       #STATE_DISCONNECTING:
         IF #disconnect.STATUS = #RESULT_JOB_START THEN
           #connectionStatus.isConnected := FALSE;
           #connectionStatus.isDisconnecting := TRUE;

         ELSIF #disconnect.STATUS = #RESULT_IDLE THEN
           #connectionStatus.isDisconnecting := TRUE;
           #disconnect.REQ := NOT #disconnect.REQ;

         ELSIF #disconnect.STATUS = #RESULT_JOB_RUNNING THEN
           #disconnect.REQ := FALSE;

         ELSIF #disconnect.STATUS = #RESULT_JOB_NOT_REQUIRED OR
           #disconnect.STATUS = #RESULT_SUCCESS
         THEN
           #disconnect.REQ := FALSE;
           #connectionStatus.isConnected := FALSE;
           #connectionStatus.isDisconnecting := FALSE;
           #connectionStatus.isDisconnected := TRUE;
           #connectionStatus.hasReceivedData := FALSE;
           #connectionStatus.hasReceivedHeader := FALSE;

           #ownInstance := 0;
           #ownSequence := 0;
           #Config.connID := 0;

           #internalState := #STATE_IDLE;
         ELSE
           // Throw error !
           //   Error from disconnecting
           #Status := W#16#8400 OR (#disconnect.STATUS AND 16#00FF);
           #disconnect.REQ := FALSE;
           #connectionStatus.isConnected := FALSE;
           #connectionStatus.isDisconnecting := FALSE;
           #connectionStatus.isDisconnected := TRUE;
           #connectionStatus.hasReceivedData := FALSE;
           #connectionStatus.hasReceivedHeader := FALSE;

           #ownInstance := 0;
           #ownSequence := 0;

           #internalState := #STATE_IDLE;
         END_IF;
       ELSE
         // Throw error !
         //   unknown internal state        
         #Status := W#16#8C00 OR (UINT_TO_WORD(#internalState) AND W#16#00FF);
     END_CASE;
   END_IF;

   #previousRequest := #REQ;
   #EnabledJ := #Enable;

   // Diagnose the connection

   #diag(ID := #connection.ID,
         RESULT := #diagStatus);

   IF #diag.STATUS = #RESULT_SUCCESS THEN
     #diag.REQ := FALSE;
     #Established := (#diagStatus.State = B#16#04);
     #Connecting := (#diagStatus.State = B#16#02) OR (#diagStatus.State = B#16#01);
   ELSIF #diag.STATUS = #RESULT_IDLE OR #diag.STATUS = #RESULT_JOB_START THEN
     #diag.REQ := TRUE;
   ELSIF #diag.STATUS = #RESULT_JOB_RUNNING THEN
     #diag.REQ := FALSE;
   ELSE
     #diag.REQ := FALSE;
     #Established := FALSE;
     #Connecting := FALSE;
   END_IF;
END_FUNCTION_BLOCK